Universal Robots URScript: Project1pick2.script

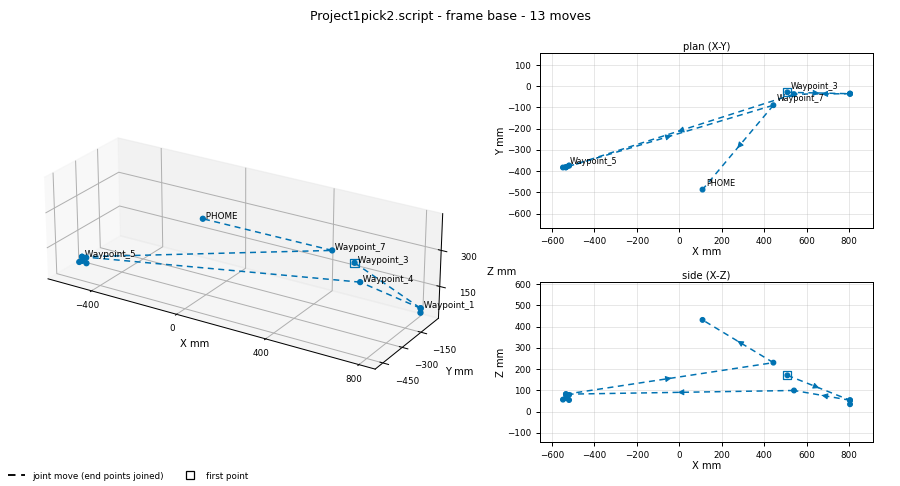
[picture p0: tool path of Project1pick2.script in frame base, 13 of 13 moves have a stored position in this frame; points joined in program order, loops and branches not executed]
def Project1pick2():
  set_tool_voltage(0)
  set_safety_mode_transition_hardness(0)
  modbus_add_signal("127.0.0.1", 255, 1, 2, "MODBUS_1", False)
  modbus_set_signal_update_frequency("MODBUS_1", 10)
  modbus_add_signal("127.0.0.1", 255, 128, 0, "atLocation", False)
  modbus_set_signal_update_frequency("atLocation", 10)
  modbus_add_signal("10.241.34.56", 1, 1009, 3, "MODBUS_2", False)
  modbus_set_signal_update_frequency("MODBUS_2", 10)
  modbus_set_runstate_dependent_choice("MODBUS_2",0)
  set_tcp(p[0.0,0.0,0.0,0.0,0.0,0.0])
  set_payload(1.0)
  step_count_de09ae77_c3e7_4e92_a6df_b707a91795b8 = 0.0
  thread Step_Counter_Thread_3807b067_43c9_469c_8c0c_342ccaebb5c8():
    while (True):
      step_count_de09ae77_c3e7_4e92_a6df_b707a91795b8 = step_count_de09ae77_c3e7_4e92_a6df_b707a91795b8 + 1.0
      sync()
    end
  end
  run Step_Counter_Thread_3807b067_43c9_469c_8c0c_342ccaebb5c8()
  set_standard_analog_input_domain(0, 1)
  set_standard_analog_input_domain(1, 1)
  set_tool_analog_input_domain(0, 0)
  set_tool_analog_input_domain(1, 0)
  set_analog_outputdomain(0, 0)
  set_analog_outputdomain(1, 0)
  set_input_actions_to_default()
  set_gravity([0.0, 0.0, 9.82])
  $ 1 "Robot Program"
  $ 2 "Set DO[0]=Off"
  set_standard_digital_out(0, False)
  $ 3 "Set DO[1]=Off"
  set_standard_digital_out(1, False)
  $ 4 "MoveJ"
  $ 5 "Waypoint_3" "breakAfter"
  movej(get_inverse_kin(p[.508862438714, -.028636304084, .170727470542, -2.196986498727, -2.240712990886, -.005196109745], qnear=[-3.414398733769552, -1.332874600087301, 2.0206899642944336, -2.2571328322040003, -1.5662038961993616, -3.43410832086672]), a=1.3962634015954636, v=1.0471975511965976)
  $ 6 "Waypoint_1" "breakAfter"
  movej(get_inverse_kin(p[.804111907576, -.035220184417, .053433598759, 2.199611793378, -2.238165059301, .005546403717], qnear=[-3.3208892981158655, -0.5748861471759241, 1.064873218536377, -2.061659638081686, -1.575683895741598, -0.16192418733705694]), a=1.3962634015954636, v=1.0471975511965976)
  $ 7 "Waypoint_2" "breakAfter"
  movej(get_inverse_kin(p[.804119060719, -.035218489685, .034566446929, 2.199697911885, -2.238226675761, .005681660345], qnear=[-3.3208892981158655, -0.5503733793841761, 1.0696830749511719, -2.0911129156695765, -1.5756481329547327, -0.161936108266012]), a=1.3962634015954636, v=1.0471975511965976)
  $ 8 "Wait: 0.5"
  sleep(0.5)
  $ 9 "Set DO[0]=On"
  set_standard_digital_out(0, True)
  $ 10 "Wait: 0.5"
  sleep(0.5)
  $ 11 "Waypoint_1" "breakAfter"
  movej(get_inverse_kin(p[.804111907576, -.035220184417, .053433598759, 2.199611793378, -2.238165059301, .005546403717], qnear=[-3.3208892981158655, -0.5748861471759241, 1.064873218536377, -2.061659638081686, -1.575683895741598, -0.16192418733705694]), a=1.3962634015954636, v=1.0471975511965976)
  $ 12 "Waypoint_4" "breakAfter"
  movej(get_inverse_kin(p[.540197777671, -.037260164018, .099373431343, 2.199778521711, -2.238179926002, .005608851214], qnear=[-3.4126973787890833, -1.142893139516012, 1.991396427154541, -2.420718495045797, -1.5754922072040003, -0.25380260149110967]), a=1.3962634015954636, v=1.0471975511965976)
  $ 13 "Waypoint_5" "breakAfter"
  movej(get_inverse_kin(p[-.534594951750, -.381840126668, .081963528749, .017860233004, 3.136760395605, .000051951932], qnear=[-5.830136273301129, -0.9117897192587732, 1.6380839347862437, -2.2927888075529985, -1.5687087217774156, -1.1063642128392033]), a=1.3962634015954636, v=1.0471975511965976)
  $ 14 "Waypoint_6" "breakAfter"
  movej(get_inverse_kin(p[-.548456452039, -.382853299182, .056301346735, .017990850984, 3.136891006613, .000060958856], qnear=[-5.83793351451029, -0.8499568144427698, 1.607193946838379, -2.323831383381979, -1.5688045660602015, -1.1140783468829554]), a=1.3962634015954636, v=1.0471975511965976)
  $ 15 "Wait: 0.5"
  sleep(0.5)
  $ 16 "Set DO[0]=Off"
  set_standard_digital_out(0, False)
  $ 17 "Wait: 0.5"
  sleep(0.5)
  $ 18 "Waypoint_8" "breakAfter"
  movej(get_inverse_kin(p[-.534540484566, -.381876234414, .064009700672, .017728478314, 3.136698426389, .000059145130], qnear=[-5.830052379761644, -0.8831418196307528, 1.645329475402038, -2.3286240736559325, -1.5686848799349669, -1.1063642128392055]), a=1.3962634015954636, v=1.0471975511965976)
  $ 19 "Wait: 0.5"
  sleep(0.5)
  $ 20 "Set DO[0]=On"
  set_standard_digital_out(0, True)
  $ 21 "Loop force()≤50"
  while ( force () <= 50):
    $ 22 "Waypoint_9" "breakAfter"
    movej(get_inverse_kin(p[-.519780689689, -.373985338934, .054327847562, .019424530609, 3.137027803560, -.001235226939], qnear=[-5.8311320880994995, -0.8951008955584818, 1.7039799690245099, -2.375984017048472, -1.5680974165554709, -1.1063642128392055]), a=1.3962634015954636, v=1.0471975511965976)
  end
  $ 23 "Wait: 0.5"
  sleep(0.5)
  $ 24 "Set DO[1]=On"
  set_standard_digital_out(1, True)
  $ 25 "Wait: 2.5"
  sleep(2.5)
  $ 26 "Waypoint_10" "breakAfter"
  movej(get_inverse_kin(p[-.519788772823, -.373980861009, .078734357621, .019443546999, 3.137086260514, -.001280621733], qnear=[-5.831144068633163, -0.9359849135028213, 1.6951265335082208, -2.3263118902786806, -1.5680974165549806, -1.1063642128392055]), a=1.3962634015954636, v=1.0471975511965976)
  $ 27 "Set DO[0]=Off"
  set_standard_digital_out(0, False)
  $ 28 "Wait: 0.5"
  sleep(0.5)
  $ 29 "Waypoint_5" "breakAfter"
  movej(get_inverse_kin(p[-.534594951750, -.381840126668, .081963528749, .017860233004, 3.136760395605, .000051951932], qnear=[-5.830136273301129, -0.9117897192587732, 1.6380839347862437, -2.2927888075529985, -1.5687087217774156, -1.1063642128392033]), a=1.3962634015954636, v=1.0471975511965976)
  $ 30 "Waypoint_7" "breakAfter"
  movej(get_inverse_kin(p[.442980114422, -.089507488081, .230504473717, -3.141481723853, .017852609412, -.007739575080], qnear=[-3.5852969328496025, -1.554119888936115, 2.094259262086275, -2.1153762976338566, -1.5686605612457267, -2.0031302610966035]), a=1.3962634015954636, v=1.0471975511965976)
  $ 31 "PHOME" "breakAfter"
  movej(get_inverse_kin(p[.109136814233, -.486931774420, .431877607004, -.000028285966, 3.141434322887, -.000393683479], qnear=[1.5707424879074097, -1.5707839171039026, 1.5707969665527344, -1.5710600058185022, -1.5706380049334925, -7.18275653284195E-5]), a=1.3962634015954636, v=1.0471975511965976)
end
